FUNCTION_BLOCK INTERNAL FB_ErrorState IMPLEMENTS I_State
VAR
	pMachine 			: POINTER TO FB_MACHINE;
END_VAR

METHOD PUBLIC Check
THIS^.ResetContactors();
THIS^.ResetTimer();
END_METHOD

PROPERTY Description : STRING
GET
Description := 'ERROR';
END_GET
END_PROPERTY

METHOD PUBLIC FB_init
VAR_INPUT
	bInitRetains : BOOL; // if TRUE, the retain variables are initialized (warm start / cold start)
	bInCopyCode : BOOL;  // if TRUE, the instance afterwards gets moved into the copy code (online change)
	
	pMachine : POINTER TO FB_MACHINE;
END_VAR
THIS^.pMachine := pMachine;
END_METHOD

METHOD PUBLIC PressButton
END_METHOD

METHOD PUBLIC PressDischarge
END_METHOD

METHOD PUBLIC Reset
THIS^.pMachine^.SetState(THIS^.pMachine^.DisconnectedState);
END_METHOD

METHOD PUBLIC ResetContactors
VAR
	nIdx					: INT := 0; 
	bBypassContactors		: ARRAY[0..1] OF BOOL; 
	bMainContactors			: ARRAY[0..1] OF BOOL; 
END_VAR
FOR nIdx := 0 TO 1 BY 1 DO 
	bBypassContactors[nIdx] := FALSE;
	bMainContactors[nIdx] := FALSE; 
END_FOR

THIS^.pMachine^.BypassContactors := bBypassContactors; // Reset every contactor 
THIS^.pMachine^.MainContactors := bMainContactors;
END_METHOD

METHOD PUBLIC ResetTimer
THIS^.pMachine^.charge_TON.IN := FALSE;
END_METHOD

METHOD PUBLIC Stop
END_METHOD

METHOD PUBLIC TimerDone
END_METHOD

END_FUNCTION_BLOCK

(* stored: Version 1.1.0.1, ProductVersion 3.1.4024.12
   POU FB_ErrorState: Id {3bd6edf8-9c55-4d99-bb9c-5733c675ad2b}, SpecialFunc None
   Method Check: Id {18a76895-891c-46c4-9487-96ee095848a3}
   Property Description: Id {6c4618e2-c37c-426d-b181-27b2e932bd77}
   Get Get: Id {20bf90f8-44dd-46b4-9988-868820b5b162}
   Method FB_init: Id {3a331c39-76aa-4ddd-9ff8-92c2148a6774}
   Method PressButton: Id {7331e6e2-e84f-4f11-be2c-061ff44361dd}
   Method PressDischarge: Id {e9c3d438-35f9-4640-8bda-eb6be60a5be5}
   Method Reset: Id {f6eab5b7-2715-4b49-8c8c-4676f5372220}
   Method ResetContactors: Id {90578b5a-f601-4b5e-95d8-9d801b8df047}
   Method ResetTimer: Id {efa99194-c307-4935-a5b5-d33cb2102d16}
   Method Stop: Id {ae111b00-ee49-4409-b4b1-c240c73646e8}
   Method TimerDone: Id {a5dd5c99-c1e0-4112-8364-4fb70dfcbe7b} *)
